// Enumerator containing general function of module
{attribute 'qualified_only'}
{attribute 'strict'}
{attribute 'to_string'}
TYPE E_Function :
(
	None,
	eSlider,
	eSliderWithGripper,
	eXYMover
);
END_TYPE

(* stored: Version 1.1.0.1, ProductVersion 3.1.4024.12
   DUT E_Function: Id {175e4159-9dd0-4f87-a565-d2b736e86ca1} *)
